{attribute addProperty BoxType "ELX5151-0000-0016"}
{attribute addProperty Id "StatusAT %I*Status_F20CBC021620Counter_valueAT %I*UINT16217"}
{attribute addProperty CRC "2869953728"}
{attribute addProperty SizeInBites "32"}
{attribute addProperty SizeInBytes "4"}
TYPE ENC_Status_compact_AB1004C0 :
STRUCT
	{attribute addProperty Name "Status"}
	Status AT %I* : Status_F20CBC02;
	{attribute addProperty Name "Counter_value"}
	Counter_value AT %I* : UINT;
END_STRUCT
END_TYPE

(* stored: Version 1.2.0.0, ProductVersion 3.1.4024.9
   DUT ENC_Status_compact_AB1004C0: Id {6afe1a28-abe3-40b8-96a8-61401398d443} *)
